/// This function block is a container for all linked units that are used by this unit.
/// Linked units can be addressed through their individual interface.
FUNCTION_BLOCK ScriblyLinkedUnit EXTENDS ScriblyContainer
VAR_INPUT

{attribute '__ZwPlcUnitEquipmentDeclaration__'} // Do not remove this attribute! It is used for code generation.
END_VAR

IF _isInitialized
THEN
  RETURN;
END_IF

{attribute '__ZwPlcUnitEquipmentImplementation__'} // Do not remove this attribute! It is used for code generation.

_isInitialized := TRUE;

END_FUNCTION_BLOCK

(* stored: Version 1.1.0.1
   POU ScriblyLinkedUnit: Id {274c1301-c80f-43b4-8e85-f04b22233deb}, SpecialFunc None *)
